(* Schneider Machine Expert - Basic project TransportRoutController, file version 2.9.0.0 *)
(* ProjectInformations: Name=New project *)

HARDWARE
  Cpu 0: TM221CE16R
  EthernetConfiguration: NetworkName=M221, IpAllocationMode=FixedAddress, IpAddress=192.168.50.50, SubnetMask=255.255.255.0
  SerialLineConfiguration: Baud=Baud19200, Parity=ParityEven, DataBits=DataBits8, StopBits=StopBits1, PhysicalMedium=PhysicalMediumRs485, SlaveId=1, Addressing=SlaveAddressing
  MastTask: UsePeriodScanMode=false, PeriodScan=100
  FastTask: Period=255
  CpuBehavior: StartingMode=StartAsPreviousState, AutoSaveRamOnEeprom=true, WatchdogPeriod=250

SYMBOLS  (address, symbol, comment, settings)
  %M0       PART_AVAILABLE
  %MW0      WORKPIECE_COUNTER
  %I0.0     LIMIT_SWITCH_SLIDER
  %I0.1     LIGHT_BARRIER_BELT
  %I0.2     LIGHT_BARRIER_PALLET_TOP
  %I0.3     LIGHT_BARRIER_PALLET_BOTTOM
  %Q0.0     MOTOR_SLIDER_PUSHER
  %Q0.1     MOTOR_BELT
  %Q0.2     VALVE_SEPARATOR

POU New POU
  (* SectionNumber=1 *)

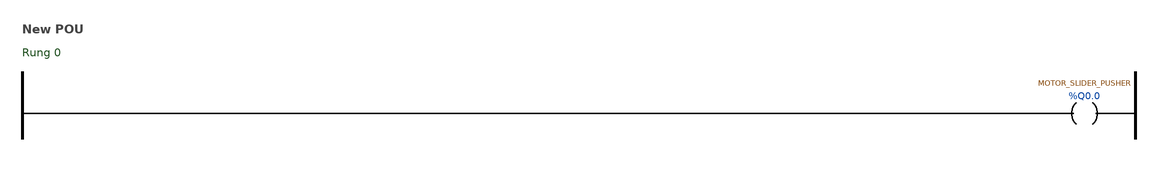

// Rung 0
  LD 1
  ST %Q0.0                (* MOTOR_SLIDER_PUSHER *)
  // as ST:
  //   MOTOR_SLIDER_PUSHER := TRUE;
